// TIA Portal project "Project3(HMI)" (V20)

(* hardware
DEVICE "S7-1500/ET200MP station_1"  S7-1500 station
   slot 0: "Rail_0"  Rack  6ES7 590-1***0-0AA0
   slot 1: "Controller"  CPU 1512C-1 PN  6ES7 512-1CK00-0AB0  V2.9
      slot 3: "CPU display_1"  6ES7591-1AA00-0AA0
      slot 32768: "PROFINET interface_1"  X1
         slot 32769: "Port_1"  X1 P1
         slot 32770: "Port_2"  X1 P2
      slot 34817: "Virtual CP interface port_1"  Virtual CP interface port  Virtual CP interface port
DEVICE "Touchpanel"  TP700 Comfort
   slot 0: "Touchpanel"  TP700 Comfort  6AV2 124-0GC01-0AX0  17.0.0.0
   slot 1: "HMI_RT_1"  TP700 Comfort  6AV2 124-0GC01-0AX0  17.0.0.0
   slot 5: "Touchpanel.IE_CP_1"  PROFINET Interface  17.0.0.0
      slot 1: "PROFINET Interface_1"  PROFINET Interface
         slot 1: "Port_1"  Port
         slot 2: "Port_2"  Port
   slot 7: "Touchpanel.MPI/DP_CP_1"  MPI/DP Interface  17.0.0.0
*)

// ===== PLC "Controller"  CPU 1512C-1 PN =====

VAR_GLOBAL   // PLC tag table "Default tag table"
   "Analog Input" AT %IW0 : Int;
   "Analog Output" AT %QW0 : Int;
   "Empty Tank" AT %I10.0 : Bool;
   "Fill In Tank" AT %I10.1 : Bool;
   "LED Indicator" AT %Q4.0 : Bool;
END_VAR

DATA_BLOCK "HMI Communication"   // DB1
{ S7_Optimized_Access := 'TRUE' }
VERSION : 0.1
   VAR
      "Analog Input" : Int;
      "Analog Output" : Int;
      "Empty Tank" : Bool;
      "Fill In Tank" : Bool;
      "LED Indicator" : Bool;
   END_VAR
BEGIN
END_DATA_BLOCK

ORGANIZATION_BLOCK "Main"   // OB1, LAD, ProgramCycle
TITLE = "Main Program Sweep (Cycle)"
{ S7_Optimized_Access := 'TRUE' }
VERSION : 0.1
   VAR_INPUT
      Initial_Call : Bool;   // Initial call of this OB
      Remanence : Bool;   // =True, if remanent data are available
   END_VAR
BEGIN

REGION Network 1
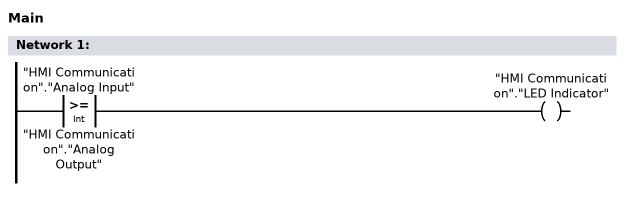
   RUNG wire#powerrail
      { S7_Templates := "SrcType := Int" } GE_Contact(in1 := "HMI Communication"."Analog Input", in2 := "HMI Communication"."Analog Output")
      Coil( "HMI Communication"."LED Indicator" )
   END_RUNG
   // the same network as SCL:
   "HMI Communication"."LED Indicator" := "HMI Communication"."Analog Input" >= "HMI Communication"."Analog Output";
END_REGION
END_ORGANIZATION_BLOCK

(* ===== HMI "HMI_RT_1" =====
system functions are stored by id; their names below are inferred from use
connection "HMI_Connection_1": ETHERNET, S7_1500_OMS

HMI tags "Default tag table"
   "Fill In Tank" : Bool = PLC "HMI Communication"."Fill In Tank" AT %I10.1, 100 ms
   "Empty Tank" : Bool = PLC "HMI Communication"."Empty Tank" AT %I10.0, 100 ms
   "LED Indicator" : Bool = PLC "HMI Communication"."LED Indicator" AT %Q4.0, 100 ms
   "Analog Input" : Int = PLC "HMI Communication"."Analog Input" AT %IW0, 100 ms
   "Analog Output" : Int = PLC "HMI Communication"."Analog Output" AT %QW0, 100 ms

screen "Root screen" 800x420, template "Template_1"
   on GenerateScreen: SetTag("@DiagnosticsIndicatorTag", 1)
   TextField "HmiScreenItemData" at 80,166 size 640x25; Text 'Welcome to HMI_1 (TP700 Comfort)!'
   Button "Button_1" at 16,256 size 156x77; TextOff 'Fill In Tank'
      on Press: function_b14e0dd5("Fill In Tank", 0)
   Bar "Bar_1" at 635,112 size 124x232; MinimumValue -20000; MaximumValue 20000
      ProcessValue <- "Analog Input"
   Slider "Slider_1" at 92,9 size 441x146; Caption 'SIMATIC'
      ProcessValue <- "Analog Output"
   Circle "Circle_1" at 484,278 size 48x48
      Appearance <- "LED Indicator"
   Switch "Switch_1" at 225,242 size 163x93; CaptionText 'Switch'; TextOff 'Empty Tank'; TextOn 'Emptying tank'
      ProcessValue <- "Empty Tank"

Template "Template_1" 800x420
   Button "Exit" at 720,360 size 78x58; TextOff 'Exit'; PictureOff "ExitRuntime_TP700_Comfort_TR"; PictureOn "ExitRuntime_TP700_Comfort_TR"
      on Release: StopRuntime(0)
   Button "Template_Button" at 640,360 size 78x58; TextOff 'Text'
   Button "Template_Button_1" at 560,360 size 78x58; TextOff 'Text'
   Button "Template_Button_2" at 480,360 size 78x58; TextOff 'Text'
   Button "Template_Button_3" at 400,360 size 78x58; TextOff 'Text'
   Button "Template_Button_4" at 321,360 size 78x58; TextOff 'Text'
   Button "Template_Button_5" at 241,360 size 78x58; TextOff 'Text'
   Button "Template_Button_6" at 161,360 size 78x58; TextOff 'Text'
   Button "Template_Button_7" at 81,360 size 78x58; TextOff 'Text'
   Button "Start screen" at 1,360 size 78x58; TextOff 'Start screen'; PictureOff "NavigateHome_TP700_Comfort_TR"; PictureOn "NavigateHome_TP700_Comfort_TR"
      on Release: ActivateScreen("Root screen", 0)
*)